// TwinCAT 3 PLC project TCP_IP_1
// ProgramVersion: 3.1.4023.0
// libraries:
//   Tc2_Standard, * (Beckhoff Automation GmbH)
//   Tc2_System, * (Beckhoff Automation GmbH)
//   Tc2_TcpIp, * (Beckhoff Automation GmbH)
//   Tc3_Module, * (Beckhoff Automation GmbH)
// project tree:
//   / PlcTask.TcTTO
//   POUs/ Client.TcPOU, MAIN.TcPOU, Server.TcPOU
// (motion and I/O tree: see PLC project ftp)
// real-time tasks:
//   TASK PlcTask: cycle T#10ms, priority 20, ADS port 350
//   TASK PlcTask1: cycle T#10ms, priority 21, ADS port 351
//   TASK PlcTask2: cycle T#10ms, priority 22, ADS port 352
//   TASK PlcTask3: cycle T#10ms, priority 23, ADS port 353
//   TASK PlcTask4: cycle T#10ms, priority 24, ADS port 354
//   TASK PlcTask5: cycle T#10ms, priority 25, ADS port 355
//   TASK PlcTask6: cycle T#10ms, priority 26, ADS port 356

CONFIGURATION TCP_IP_1
    RESOURCE PLC ON TwinCAT3
        TASK PlcTask(INTERVAL := T#10ms, PRIORITY := 21);
        PROGRAM MAIN WITH PlcTask : MAIN;
    END_RESOURCE
END_CONFIGURATION

// ---- POUs/MAIN.TcPOU
PROGRAM MAIN

VAR
    hServer         : T_HSERVER; 
END_VAR

Server(hServer := hServer);
Client();

END_PROGRAM

// ---- POUs/Server.TcPOU
PROGRAM Server

VAR_IN_OUT
    hServer         : T_HSERVER; 
END_VAR

VAR_INPUT
	CLOSE_CONNECTION : BOOL := FALSE;
END_VAR

VAR
	FB_ServerClientConnection: FB_ServerClientConnection;
	FB_SocketSend: FB_SocketSend;
	FB_SocketCloseAll: FB_SocketCloseAll;
	
	DATA 	   : BYTE := 1;
	pSrc       : POINTER TO BYTE := ADR(DATA);
END_VAR

// The function F_CreateServerHnd is used to initialise/set the internal parameters of a server handle variable hServer.
// The server handle is then transferred to the instances of the FB_ServerClientConnection function block via VAR_IN_OUT. 
F_CreateServerHnd(
	sSrvNetID:= '', 
	sLocalHost:= '', 
	nLocalPort:= 200, 
	nMode:= LISTEN_MODE_CLOSEALL OR CONNECT_MODE_ENABLEDBG, 
	bEnable:= TRUE, 
	hServer:= hServer);

FB_ServerClientConnection(
	hServer:= hServer, 
	eMode:= eACCEPT_ALL,
	sRemoteHost:= '',
	nRemotePort:= 200,
	bEnable:= TRUE, 
	tReconnect:= T#1S);

IF FB_ServerClientConnection.eState = eSOCKET_CONNECTED THEN
	FB_SocketSend(
	sSrvNetId:= '', 
	hSocket:= FB_ServerClientConnection.hSocket, 
	cbLen:= 8, 
	pSrc:= pSrc, 
	bExecute:= TRUE, 
	tTimeout:= T#10S);
END_IF
	
FB_SocketCloseAll(
	sSrvNetId:= '', 
	bExecute:= CLOSE_CONNECTION, 
	tTimeout:= T#1S);

END_PROGRAM

// ---- POUs/Client.TcPOU
PROGRAM Client

VAR
	FB_ClientServerConnection: FB_ClientServerConnection;
	FB_SocketReceive: FB_SocketReceive;
	
	FB_SocketSend:FB_SocketSend;
	fbDataExchaTON: TON;
	sFromServer: T_MaxString;
END_VAR

VAR_INPUT
	RECEIVE    : BYTE;
	pSrc       : POINTER TO BYTE := ADR(RECEIVE);
END_VAR

FB_ClientServerConnection(
	sSrvNetID:= '',				// String dat het AMS netwerk-adres van de TwinCAT TCP/IP connectie server bevat. (Local pc == empty string).
	nMode:= 0, 					// Additional Parameter flag.
	sRemoteHost:= '', 			// IP-Adres van (IPv4) van de remote server als string. (Local pc == empty string).
	nRemotePort:= 200,		    // IP-port number voor de remote server. 
	bEnable:= TRUE,				// Zolang deze INPUT = TRUE probeert het systeem een connectie aan te gaan in 'bepaalde intervallen' totdat een connectie is aangegaan.
	tReconnect:= T#1S);			// Cycle bepaalde intervallen

IF FB_ClientServerConnection.eState = eSOCKET_CONNECTED THEN
	fbDataExchaTON( IN := TRUE, PT := T#1S );

	FB_SocketReceive(
		sSrvNetId:= '', 
		hSocket:= FB_ClientServerConnection.hSocket, 
		cbLen:= 8, 
		pDest:= pSrc, 
		bExecute:= TRUE, 
		tTimeout:= T#10S);
END_IF

END_PROGRAM
